Fanuc KAREL source: kt00342.KL

-- PROVISIONAL review KL for V770-1; original PC SHA256 5e5b600e72ee43c74889baf060100e96195b27978f3a79f865cbb18f6bef101e
-- Incomplete behavior may be omitted. Consult companion uncertainty JSON. Do not deploy.
PROGRAM KT00342
%NOLOCKGROUP
VAR
  OUT : BOOLEAN
-- UNRESOLVED_DECL Y1 type=002018
-- UNRESOLVED_DECL H2 type=002017
BEGIN
  -- UNRESOLVED_PC offsets 5-19; opcodes 2E,22,9D,33,B2
  -- UNRESOLVED_PC offsets 24-38; opcodes 2E,22,9D,33,B4
  -- UNRESOLVED_PC offsets 43-68; opcodes 22,9D,33,B1,22,9D,33,B3,59,23
  -- UNRESOLVED_PC offsets 73-77; opcodes 7F
END KT00342
